FUNCTION_BLOCK FB_IOFileReadWrite
VAR_IN_OUT
	readBuff:ARRAY [*] OF ST_DataFmtBase;
END_VAR
VAR_INPUT
	sFileName:T_MaxString:='C:\CsvFilePath\csvfile.csv';//'Hard Disk\CsvFilePath\csvfile.csv'
	bRead:BOOL;
	sTxtHead:STRING:='GROUP,NUM,ENG,CHN,NO USE';
END_VAR
VAR_OUTPUT
	bBusy:BOOL;
	bDone:BOOL;
	bError:BOOL;
	nErrid:UDINT;
END_VAR
VAR
	fbFileOpen:FB_FileOpen;
	fbFileClose:FB_FileClose;
	fbFileGets:FB_FileGets;
	fbReader:FB_CSVMemBufferReader;
	hFile:UINT:= 0;
	
	sReadLine:STRING(255);
	bReadEOF:BOOL;
	nReadCount:DINT;
	
	nStepRead:UINT;
	nReadBuffMin:DINT;
	nReadBuffMax:DINT;
	nReadBuffLen:DINT;
END_VAR


nReadBuffMin:=LOWER_BOUND(readBuff,1);//获取不定长数组的最小下标
nReadBuffMax:=UPPER_BOUND(readBuff,1);//获取不定长数组的最大下标
nReadBuffLen:=nReadBuffMax-nReadBuffMin+1;//获取数组有效长度

readCSV();

//

METHOD PRIVATE createDir : BOOL
VAR
	sPathNameTemp	: T_MaxString := 'C:\TwinCAT\Data.txt';
	sDriveTemp		: STRING(3);
	sDirTemp		: T_MaxString;
	sFileNameTemp	: T_MaxString;
	sExtTemp		: T_MaxString;
	bSuccess		: BOOL;
	fbCreateDir		: FB_CreateDir;
	sFileDirTemp	: T_MaxString;
END_VAR
sPathNameTemp:=sFileName;
bSuccess := F_SplitPathName(sPathName:= sPathNameTemp,
						sDrive:= sDriveTemp,
						sDir:= sDirTemp,
						sFileName:= sFileNameTemp,
						sExt:= sExtTemp );
IF bSuccess THEN
	bSuccess:=FALSE;
	IF LEFT(sDirTemp,LEN(sDirTemp)-1)<>'' THEN
		sFileDirTemp:=CONCAT(STR1:=sDriveTemp,STR2:=LEFT(sDirTemp,LEN(sDirTemp)-1));
		fbCreateDir(
			sNetId:= , 
			sPathName:= sFileDirTemp, 
			ePath:= PATH_GENERIC, 
			bExecute:= TRUE, 
			tTimeout:= , 
			bBusy=> , 
			bError=> , 
			nErrId=> );
	END_IF
END_IF
fbCreateDir(
	sNetId:= , 
	sPathName:= , 
	ePath:= , 
	bExecute:= FALSE, 
	tTimeout:= , 
	bBusy=> , 
	bError=> , 
	nErrId=> );
END_METHOD

METHOD PRIVATE readCSV : BOOL
VAR_INPUT
END_VAR
VAR
	nTemp_readCSV:INT;
	sGetValue_temp:STRING(255);
	bRtn:BOOL;
	nTemp1:INT;
END_VAR
DEFAULT_CSV_FIELD_SEP:= 16#2C;  //配置CSV文件的分割符，16#2C表明各个参数之间是用逗号分隔的。

CASE nStepRead OF
	0:
		IF bRead THEN
			bRead:=FALSE;
			bBusy:=TRUE;
			bDone:=FALSE;
			bError:=FALSE;
			nErrid:=0;
			
			nReadCount:=nReadBuffMin;			
			MEMSET(readBuff,0,TO_UDINT(SIZEOF(readBuff[nReadCount])*nReadBuffLen));//清空内存
			nStepRead:=100;
		END_IF
	100:
		fbFileOpen(bExecute:=FALSE);
		nStepRead:=nStepRead+10;
	110:
		fbFileOpen(
			sNetId:= , 
			sPathName:= sFileName, 
			nMode:= FOPEN_MODEREAD OR FOPEN_MODETEXT, 
			ePath:= PATH_GENERIC, 
			bExecute:= TRUE, 
			tTimeout:= , 
			bBusy=> , 
			bError=> , 
			nErrId=> , 
			hFile=> hFile);
		IF NOT fbFileOpen.bBusy THEN
			IF NOT fbFileOpen.bError THEN
				nStepRead:=nStepRead+10;
			ELSE
				nErrid:=fbFileOpen.nErrId;
				nStepRead:=60000;//Error
			END_IF
		END_IF
	120:
		fbFileGets(bExecute:=FALSE);
		IF nReadCount>nReadBuffMax THEN
			nStepRead:=150;
		ELSE
			nStepRead:=nStepRead+10;
		END_IF
	130:
		fbFileGets(
			sNetId:= , 
			hFile:= hFile, 
			bExecute:= TRUE, 
			tTimeout:= , 
			bBusy=> , 
			bError=> , 
			nErrId=> , 
			sLine=> sReadLine, 
			bEOF=> bReadEOF);
		IF NOT fbFileGets.bBusy THEN
			IF NOT fbFileGets.bError THEN
				sReadLine:=CONCAT(STR1:=sReadLine,STR2:='$R$L');
				nStepRead:=nStepRead+10;
			ELSE
				nErrid:=fbFileGets.nErrId;
				nStepRead:=60000;//Error
			END_IF
		END_IF
	140:
		IF ''<>sTxtHead AND FIND(sReadLine,sTxtHead)>0 THEN
			nStepRead:=120;
			RETURN;
		END_IF
		nTemp1:=0;
		fbReader.eCmd:=eEnumCmd_First;(* Read first field value *)
		FOR nTemp_readCSV:=0 TO 3 DO
			fbReader(
				eCmd:= , 
				pBuffer:= ADR(sReadLine), 
				cbBuffer:= SIZEOF(sReadLine), 
				bOk=> , 
				getValue=> sGetValue_temp, 
				pValue=> , 
				cbValue=> , 
				bCRLF=> , 
				cbRead=> );
			IF fbReader.bOk THEN
				fbReader.eCmd:=eEnumCmd_Next;
				CASE nTemp_readCSV OF 
					0:
						readBuff[nReadCount].nGroup:=TO_DINT(sGetValue_temp);
					1:
						readBuff[nReadCount].nNumber:=TO_DINT(sGetValue_temp);
					2:
						readBuff[nReadCount].sTxt_ENG:=sGetValue_temp;
					3:
						bRtn:=UTF8_TO_WSTRING(ADR(readBuff[nReadCount].sTxt_CHN),ADR(sGetValue_temp),SIZEOF(sGetValue_temp));
						IF NOT bRtn OR ""=readBuff[nReadCount].sTxt_CHN THEN
							readBuff[nReadCount].sTxt_CHN:=TO_WSTRING(readBuff[nReadCount].sTxt_ENG);
						END_IF
				END_CASE
				nTemp1:=nTemp_readCSV;
			END_IF
		END_FOR
		IF NOT bReadEOF THEN
			nReadCount:=nReadCount+1;
			nStepRead:=120;
		ELSE
			nStepRead:=nStepRead+10;
		END_IF
	150:
		nStepRead:=50000;//Done

 //Done
	50000:
		fbFileOpen(bExecute:=FALSE);
		fbFileGets(bExecute:=FALSE);
		fbFileClose(bExecute:=FALSE);
		nStepRead:=nStepRead+10;
	50010:
		fbFileClose(
			sNetId:= , 
			hFile:= hFile, 
			bExecute:= TRUE, 
			tTimeout:= , 
			bBusy=> , 
			bError=> , 
			nErrId=> );
		IF NOT fbFileClose.bBusy THEN
			nStepRead:=nStepRead+10;
		END_IF
	50020:
		fbFileClose(bExecute:=FALSE);
		bBusy:=FALSE;
		bDone:=TRUE;
		bError:=FALSE;
		nStepRead:=0;
 //Error
	60000:
		fbFileOpen(bExecute:=FALSE);
		fbFileGets(bExecute:=FALSE);
		fbFileClose(bExecute:=FALSE);
		nStepRead:=nStepRead+10;
	60010:
		fbFileClose(
			sNetId:= , 
			hFile:= hFile, 
			bExecute:= TRUE, 
			tTimeout:= , 
			bBusy=> , 
			bError=> , 
			nErrId=> );
		IF NOT fbFileClose.bBusy THEN
			nStepRead:=nStepRead+10;
		END_IF
	60020:
		fbFileClose(bExecute:=FALSE);
		bBusy:=FALSE;
		bDone:=FALSE;
		bError:=TRUE;
		nStepRead:=0;
END_CASE
END_METHOD

END_FUNCTION_BLOCK

(* stored: Version 1.1.0.1, ProductVersion 3.1.4024.4
   POU FB_IOFileReadWrite: Id {3e1929ed-bbf4-486e-b54a-b4385b8322cb}, SpecialFunc None
   Method createDir: Id {1c77f885-8046-4544-99dd-9f2e6296f85d}
   Method readCSV: Id {b1f516e6-3969-4acc-8792-2ca7d928adb9} *)
